
// ===== library types =====

TYPE "LHTTP_typeTLS"
   STRUCT
      validateServerIdentity : Bool;   // Validate the subjectAlternateName in the X.509-V3 certificate of the server to check the identity of the server
      serverCert : UDInt;   // ID of the X.509-V3 certificate (usually a CA certificate) that is used by the TLS client to validate the TLS server authentication. If this parameter is 0, the TLS client uses all (CA) certificates currently loaded in the client certificate store to validate the server authentication.
      clientCert : UDInt;   // ID of own X.509 V3 certificate
   END_STRUCT;
END_TYPE

// folder: GET

FUNCTION_BLOCK "LHTTP_Get"   // FB5, SCL
{ S7_Optimized_Access := 'TRUE' }
AUTHOR : AV
FAMILY : NET
VERSION : 0.1
   VAR_INPUT
      execute : Bool;   // Send HTTP request
      hwID : HW_ANY := 64;   // Hardware ID of Ethernet interface
      connID : CONN_OUC := 1;   // Unique connection ID
      url : String;   // URL, i.e. "http://www.siemens.com/simatic"
      data : String;   // Optional query parameters that are appended to URL, i.e. "lang=en&q=simatic"
      tls : "LHTTP_typeTLS";   // TLS certificates for secure connections (HTTPS), leave open for non-secure connections (HTTP)
   END_VAR
   VAR_OUTPUT
      done : Bool;   // HTTP request finished
      busy : Bool;   // Function is busy
      error : Bool;   // An error occured
      statusID : USInt;   // Specifies the source of the error
      status : Word;   // Specifies the error
      responseCode : UInt;   // HTTP response code
      length : UDInt;   // Length of received data
   END_VAR
   VAR_IN_OUT
      responseData : Array[*] of Char;   // Data received from HTTP server
   END_VAR
   VAR
      instTSend : TSEND_C;   // Instance of TSEND_C
      instTRcv : TRCV;   // Instance of TRCV
      instTimeout : TON_TIME;   // Time-out
      statDone : Bool;   // Static value for output 'done'
      statBusy : Bool;   // Static value for output 'busy'
      statError : Bool;   // Static value for output 'error'
      statStatusID : USInt;   // Static value for output 'statusID'
      statStatus : Word := 16#7000;   // Static value for output 'status'
      statFBState : USInt := 0;   // Current state in state machine
      statResponseCode : UInt;   // Static value for output 'responseCode'
      statEncoding : String;   // Transfer encoding of response from HTTP server
      statContentLength : UInt;   // Content length as specified in header of response
      statChunkLen : UInt;   // Remaining length of current chunk
      statRcvdLen : UDInt;   // Sum length of received data
      statLength : UDInt;   // Static value for output 'length'
      statParam : Struct   // Connection parameters
         isQDN : Bool;
         paramQDN : TCON_QDN_SEC;   // Connection parameters in form of QDN
         paramIP : TCON_IP_V4_SEC;   // Connection parameters in form of IP address
      END_STRUCT;
      statSend : Struct   // Parameters for instruction TSend_C
         connect : Bool;   // Establish and keep connection
         req : Bool;   // Send data
      END_STRUCT;
      statRequest : Struct   // GET request
         chars : Array[0..601] of Char;   // GET request (max. length: url (254) + data (254) + header (94)
         length : UInt;   // Length of GET request
      END_STRUCT;
      statTimeoutIn : Bool;   // Timeout
      statRcvBuffer : Array[0..1459] of Char;   // Temporary receive buffer; maximum segment size for TCP/IP is 1460
      statSizeRcvArray : UDInt;   // Size of receive buffer at parameter "responseData"
      statExecuteOld : Bool;   // Last cycle's value of input "execute"
   END_VAR
   VAR_TEMP
      tempLowerBound : DInt;   // Lower bound of receive buffer
      tempUrl : String;   // Copy of URL
      tempHost : String;   // Host part of URL
      tempPath : String;   // Path part of URL
      tempQuery : String;   // Query part of URL
      tempIndex : Int;   // Index for for loops
      tempPos : Int;   // General tag for positions
      tempLen : UInt;   // General tag for lengths
      tempRet : Word;   // General tag for return values
      tempString : String;   // General tag for strings
      tempExitLoop : Bool;   // Condition to exit REPEAT loop around state machine
      tempChunk : Struct   // Temporary tags for chunked encoding
         posData : UInt;   // Start position of data in current packet
         lenData : UInt;   // Length of data in current packet
         exitLoop : Bool;   // Condition to exit loop
      END_STRUCT;
   END_VAR
   VAR CONSTANT
      STATUS_DONE : Word := 16#0000;   // Job finished without errors
      STATUS_IDLE : Word := 16#7000;   // No job
      STATUS_FIRST_CALL : Word := 16#7001;   // First call after incoming new job (rising edge 'execute')
      STATUS_BUSY : Word := 16#7002;   // Intermediate call after job was started
      STATUS_BOUND_NOT_ZERO : Word := 16#8101;   // Lower bound of receive buffer is not 0
      STATUS_BUFFER_SIZE : Word := 16#8102;   // Receive buffer at parameter "responseData" too small
      STATUS_INVALID_URL : Word := 16#8103;   // Invalid URL
      STATUS_INVALID_HEADER : Word := 16#8104;   // Header of response is invalid
      STATUS_ENCODING_UNKNOWN : Word := 16#8105;   // Transfer encoding of response could not be detected or is unsupported
      STATUS_LENGTH_UNKNOWN : Word := 16#8106;   // Content length of response could not be detected
      STATUS_DECODING_FAILED : Word := 16#8107;   // Chunk encoded response could not be decoded
      STATUS_FORWARDING : Word := 16#8300;   // Server responded with forwarding message. Forwarding is not supported
      STATUS_TIMEOUT : Word := 16#8408;   // Time-out occurred
      STATUS_UNDEFINED_STATE : Word := 16#8600;   // Error due to an undefined state in state machine
      STATUS_ID_TSENDC : USInt := 1;   // Source of error is TSEND_C
      STATUS_ID_TRCV : USInt := 2;   // Source of error is TRCV
      STATUS_ID_MOVE_IDENTITY : USInt := 3;   // Source of error is MOVE_BLK_VARIANT for transfer encoding 'identity'
      STATUS_ID_MOVE_CHUNKED : USInt := 4;   // Source of error is MOVE_BLK_VARIANT for transfer encoding 'chunked'
      STATUS_ID_HTTP : USInt := 5;   // HTTP server signals error
      STATE_IDLE : USInt := 0;   // State no job
      STATE_INIT : USInt := 1;   // State initialization
      STATE_SEND : USInt := 2;   // State send request
      STATE_RCV : USInt := 3;   // State receive data
      TIMEOUT : Time := t#10s;   // Time to wait for response from server
      CRLF : String := '$R$L';   // ASCII characters for CRLF (carriage return & line feed)
      HEADER_END : String := '$R$L$R$L';   // End of HTTP header (double CRLF)
      LEN_CRLF : UInt := 2;   // Length of CRLF
   END_VAR
   // statParam.paramQDN.ConnPara.ActiveEstablished := true;
   // statParam.paramIP.ConnPara.ActiveEstablished := true;
BEGIN
   //=============================================================================
   // SIEMENS AG
   // (c)Copyright 2019
   //-----------------------------------------------------------------------------
   // Library:       LHTTP
   // Tested with:   CPU 1516-3 PN/DP V2.6
   // Engineering:   TIA Portal V15.1
   // Restrictions:  --
   // Requirements:  --
   // Functionality: Implements the HTTP GET method
   //-----------------------------------------------------------------------------
   // Change log table:
   // Version    Date         Expert in charge         Changes applied
   // 01.00.00   01.04.2019   Siemens Online Support   First released version
   //=============================================================================

   REGION INSTRUCTIONS
     IF (#statStatus <> #STATUS_IDLE) THEN // Only execute when FB is triggered to reduce system load
       // Connect and send
       IF #statParam.isQDN THEN // Call if host is a domain name
         #instTSend(REQ := #statSend.req,
                    CONT := #statSend.connect,
                    LEN := #statRequest.length,
                    CONNECT := #statParam.paramQDN,
                    DATA := #statRequest.chars);
       ELSE // Call if host is an IP address
         #instTSend(REQ := #statSend.req,
                    CONT := #statSend.connect,
                    LEN := #statRequest.length,
                    CONNECT := #statParam.paramIP,
                    DATA := #statRequest.chars);
       END_IF;

       // Receive
       #instTRcv(ID := #statParam.paramQDN.ConnPara.ID,
                 EN_R := #statFBState = #STATE_RCV,
                 LEN := 0,
                 ADHOC := true,
                 DATA := #statRcvBuffer);

       // Monitor time out
       #instTimeout(IN := #statTimeoutIn,
                    PT := #TIMEOUT);

       IF #instTimeout.Q THEN
         #statStatus := #STATUS_TIMEOUT;
       END_IF;
     END_IF;
   END_REGION

   REGION TRIGGERING
     IF (#execute = true) AND (#statExecuteOld = false) // Check if FB is triggered
       AND (#statStatus = #STATUS_IDLE)
     THEN // First call; initialize FB
       #statBusy := true;
       #statStatus := #STATUS_FIRST_CALL;
       #statFBState := #STATE_INIT;
     ELSIF (#statStatus = #STATUS_FIRST_CALL) THEN
       #statStatus := #STATUS_BUSY;
     END_IF;

     // Edge detection 'execute' input
     #statExecuteOld := #execute;
   END_REGION TRIGGERING

   IF (#statStatus = #STATUS_IDLE) THEN // Nothing to do -> End here to reduce "system load"
     RETURN;
   END_IF;

   REGION STATE_MACHINE
     // State machine is wrapped in REPEAT loop to make it possible to quickly exit state machine
     // in case of an error or to go through CASE multiple times within one cycle
     REPEAT
       #tempExitLoop := true; // Condition to exit loop is set per default

       CASE #statFBState OF // State machine of FB
         #STATE_IDLE: // No processing active (Note: this state must always be present and left empty)
           ;

         #STATE_INIT:
           REGION INIT
             // Get size of receive buffer
             #tempLowerBound := LOWER_BOUND(ARR := #responseData, DIM := 1);
             IF #tempLowerBound <> 0 THEN
               #statStatus := #STATUS_BOUND_NOT_ZERO;
               EXIT; // Exit loop immediately and output error
             ELSE
               #statSizeRcvArray := DINT_TO_UDINT(UPPER_BOUND(ARR := #responseData, DIM := 1)) + 1;
             END_IF;

             // Set connection parameters
             #statParam.paramQDN.ConnPara.InterfaceId := #hwID;
             #statParam.paramQDN.ConnPara.ID := #connID;
             #statParam.paramIP.ConnPara.InterfaceId := #hwID;
             #statParam.paramIP.ConnPara.ID := #connID;

             // Copy URL
             #tempUrl := #url;

             // Check if network protocol was specified to determine if connection should be secured
             IF #tempUrl[5] = 's' OR #tempUrl[5] = 'S' THEN // HTTPS
               #statParam.paramQDN.ActivateSecureConn := true;
               #statParam.paramQDN.ExtTLSCapabilities.%X0 := #tls.validateServerIdentity;
               #statParam.paramQDN.TLSServerCertRef := #tls.serverCert;
               #statParam.paramQDN.TLSClientCertRef := #tls.clientCert;
               #statParam.paramIP.ActivateSecureConn := true;
               #statParam.paramIP.ExtTLSCapabilities.%X0 := #tls.validateServerIdentity;
               #statParam.paramIP.TLSServerCertRef := #tls.serverCert;
               #statParam.paramIP.TLSClientCertRef := #tls.clientCert;
               // Delete network protocol from URL
               #tempUrl := DELETE(IN := #tempUrl, L := 8, P := 1);
             ELSE // HTTP
               #statParam.paramQDN.ActivateSecureConn := false;
               #statParam.paramIP.ActivateSecureConn := false;
               // Delete network protocol from URL if specified
               IF #tempUrl[5] = ':' THEN
                 #tempUrl := DELETE(IN := #tempUrl, L := 7, P := 1);
               END_IF;
             END_IF;

             // Determine if host is domain name or IP address
             #tempPos := CHAR_TO_INT(#tempUrl[1]);
             IF #tempPos >= CHAR_TO_INT('A') AND #tempPos <= CHAR_TO_INT('z') THEN // Host is a domain name
               #statParam.isQDN := true;
             ELSIF #tempPos >= CHAR_TO_INT('0') AND #tempPos <= CHAR_TO_INT('9') THEN // Host is an IP address
               #statParam.isQDN := false;
             ELSE // URL invalid
               #statStatus := #STATUS_INVALID_URL;
               EXIT; // Exit loop immediately
             END_IF;

             // Get host name and port
             #tempPos := FIND(IN1 := #tempUrl, IN2 := '/');
             IF #tempPos > 0 THEN // URL has a path after host name
               #tempHost := LEFT(IN := #tempUrl, L := #tempPos - 1);
               #tempPath := DELETE(IN := #tempUrl, L := #tempPos - 1, P := 1);
             ELSE
               #tempHost := #tempUrl;
               #tempPath := '/';
             END_IF;
             #tempPos := FIND(IN1 := #tempHost, IN2 := ':');
             IF #tempPos > 0 THEN // Port specified in URL
               #statParam.paramQDN.ConnPara.RemotePort := STRING_TO_UINT(DELETE(IN := #tempHost, L := #tempPos, P := 1));
               #statParam.paramIP.ConnPara.RemotePort := STRING_TO_UINT(DELETE(IN := #tempHost, L := #tempPos, P := 1));
               #tempHost := LEFT(IN := #tempHost, L := #tempPos - 1);
             ELSE // No port specified in URL, set default port
               IF #statParam.paramQDN.ActivateSecureConn OR #statParam.paramIP.ActivateSecureConn THEN
                 #statParam.paramQDN.ConnPara.RemotePort := 443;
                 #statParam.paramIP.ConnPara.RemotePort := 443;
               ELSE
                 #statParam.paramQDN.ConnPara.RemotePort := 80;
                 #statParam.paramIP.ConnPara.RemotePort := 80;
               END_IF;
             END_IF;

             IF #statParam.isQDN THEN // Host is a domain name
               #statParam.paramQDN.ConnPara.RemoteQDN := CONCAT(IN1 := #tempHost, IN2 := '.');
             ELSE // Host is an IP address
               #tempString := #tempHost;
               FOR #tempIndex := 1 TO 3 DO
                 #tempPos := FIND(IN1 := #tempString, IN2 := '.');
                 #statParam.paramIP.ConnPara.RemoteAddress.ADDR[#tempIndex] := UINT_TO_BYTE(STRING_TO_UINT(LEFT(IN := #tempString, L := #tempPos - 1)));
                 #tempString := DELETE(IN := #tempString, L := #tempPos, P := 1);
               END_FOR;
               #statParam.paramIP.ConnPara.RemoteAddress.ADDR[4] := UINT_TO_BYTE(STRING_TO_UINT(#tempString));
             END_IF;

             // Prepare query part of URL
             IF #data <> '' THEN // Parameter data is in use
               IF #data[1] = '?' OR #data[1] = '&' THEN
                 #tempQuery := DELETE(IN := #data, P := 1, L := 1);
               ELSE
                 #tempQuery := #data;
               END_IF;
               #tempPos := FIND(IN1 := #tempPath, IN2 := '?'); // Check if URL already contains query parameters
               IF #tempPos <> 0 THEN // URL already contains query parameters
                 #tempQuery := CONCAT(IN1 := '&', IN2 := #tempQuery); // Append query parameters with &
               ELSE // URL does not contain query parameters
                 #tempQuery := CONCAT(IN1 := '?', IN2 := #tempQuery); // Append query parameters with ?
               END_IF;
             END_IF;

             // Put together GET request
             // Strg_TO_Chars conversion is done several times to utilize maximum length of parameters url and data
             Strg_TO_Chars(Strg := CONCAT(IN1 := 'GET ', IN2 := #tempPath), // Path cannot be longer than 249 characters --> save to use CONCAT
                           pChars := 0,
                           Cnt => #tempLen,
                           Chars := #statRequest.chars);
             #tempPos := UINT_TO_INT(#tempLen);

             Strg_TO_Chars(Strg := #tempQuery,
                           pChars := #tempPos,
                           Cnt => #tempLen,
                           Chars := #statRequest.chars);
             #tempPos += UINT_TO_INT(#tempLen);

             Strg_TO_Chars(Strg := CONCAT(IN1 := ' HTTP/1.1$R$LHost: ', IN2 := #tempHost), // Host will not use all 254 characters --> save to use CONCAT
                           pChars := #tempPos,
                           Cnt => #tempLen,
                           Chars := #statRequest.chars);
             #tempPos += UINT_TO_INT(#tempLen);

             Strg_TO_Chars(Strg := '$R$LUser-Agent: SIMATIC S7-1500 (LHTTP)$R$LAccept: text/html$R$LAccept-Encoding: identity$R$LAccept-Charset: utf-8$R$L$R$L',
                           pChars := #tempPos,
                           Cnt => #tempLen,
                           Chars := #statRequest.chars);
             #statRequest.length := INT_TO_UINT(#tempPos) + #tempLen;

             #statSend.connect := true; // Connect
             #statSend.req := true; // Send request
             #statTimeoutIn := true; // Start timer
             #statFBState := #STATE_SEND;
           END_REGION

         #STATE_SEND: // Send data
           REGION SEND
             IF #instTSend.DONE THEN
               #statFBState := #STATE_RCV;
               // Stay in REPEAT loop to go directly to receive state
               // without waiting for next cycle so that no responses can be missed
               #tempExitLoop := false;
             ELSIF #instTSend.ERROR THEN
               #statStatusID := #STATUS_ID_TSENDC;
               #statStatus := #instTSend.STATUS;
             END_IF;
           END_REGION

         #STATE_RCV: // Wait for new data
           REGION RCV
             IF #instTRcv.NDR THEN

               REGION HEADER_EVAL
                 // Evaluate header if received packet is first packet
                 IF #statRcvdLen = 0 THEN
                   // Get response code
                   Chars_TO_Strg(Chars := #statRcvBuffer,
                                 pChars := 9,
                                 Cnt := 3,
                                 Strg => #tempString);
                   #statResponseCode := STRING_TO_UINT(#tempString);

                   // Exit loop immediately and output errror if response code shows errors or forwarding
                   IF #statResponseCode >= 400 THEN
                     #statStatusID := #STATUS_ID_HTTP;
                     #tempRet := ATH(IN := #tempString, N := 3, OUT => #statStatus); // Interpret response code as hexadecimal to integrate in status output
                     #statStatus := SHR(IN := #statStatus, N := 4);
                     #statStatus := 16#9000 OR #statStatus;
                     EXIT;
                   ELSIF #statResponseCode >= 300 THEN
                     #statStatus := #STATUS_FORWARDING;
                     EXIT;
                   END_IF;

                   // Get length of HTTP header
                   #tempLen := DINT_TO_UINT("LHTTP_FindStringInArray"(searchFor := #HEADER_END, searchIn := #statRcvBuffer) + LEN(#HEADER_END));

                   // Exit loop immediately and output errror if header end cannot be found
                   IF #tempLen = 0 THEN
                     #statStatus := #STATUS_INVALID_HEADER;
                     EXIT;
                   END_IF;

                   // Search header for content length
                   #tempRet := "LHTTP_ExtractStringFromArray"(textBefore := 'Content-Length: ',
                                                              textAfter := #CRLF,
                                                              extractedString => #tempString,
                                                              searchIn := #statRcvBuffer);

                   IF #tempRet = 0 THEN // Content length found
                     #statContentLength := STRING_TO_UINT(#tempString);
                     #statEncoding := 'identity';
                   ELSE // Can't detect content length, check if transfer encoding is 'chunked'
                     #tempPos := DINT_TO_INT("LHTTP_FindStringInArray"(searchFor := 'chunked', searchIn := #statRcvBuffer));

                     IF #tempPos >= 0 THEN
                       #statEncoding := 'chunked';
                     ELSE // Exit loop immediately and output error if content length nor transfer encoding can be detected
                       #statStatus := #STATUS_ENCODING_UNKNOWN;
                       EXIT;
                     END_IF;
                   END_IF;
                 END_IF;
               END_REGION

               REGION TE_IDENTITY
                 IF #statEncoding = 'identity' THEN // Transfer encoding is 'identity'
                   // Move data from buffer to output; tempLen contains header length during first packet, otherwise 0
                   #tempRet := INT_TO_WORD(MOVE_BLK_VARIANT(SRC := #statRcvBuffer,
                                                                                    COUNT := MIN(IN1 := #instTRcv.RCVD_LEN - #tempLen, IN2 := #statSizeRcvArray - #statRcvdLen), // Move as much as possible to output
                                                                                    SRC_INDEX := #tempLen,
                                                                                    DEST_INDEX := UDINT_TO_DINT(#statRcvdLen),
                                                                                    DEST => #responseData));

                   // Exit loop immediately and output error if data could not be moved
                   IF #tempRet <> 0 THEN
                     #statStatusID := #STATUS_ID_MOVE_IDENTITY;
                     #statStatus := #tempRet;
                     EXIT;
                   END_IF;

                   // Add length of received packet to sum; tempLen contains header length during first packet, otherwise 0
                   #statRcvdLen += #instTRcv.RCVD_LEN - #tempLen;

                   IF #statRcvdLen > #statSizeRcvArray THEN // Receive buffer too small
                     #statStatus := #STATUS_BUFFER_SIZE;
                     #statLength := #statContentLength; // Output required size of buffer
                   ELSIF #statRcvdLen >= #statContentLength THEN // Everything was received
                     #statStatus := #STATUS_DONE;
                     #statLength := #statRcvdLen;
                   END_IF;
                 END_IF;
               END_REGION

               REGION TE_CHUNKED
                 IF #statEncoding = 'chunked' THEN // Transfer encoding is 'chunked'

                   // Set position of chunk data
                   #tempChunk.posData := #tempLen; // tempLen contains header length during first packet, otherwise 0

                   REPEAT
                     #tempChunk.exitLoop := true; // Condition to exit loop is set per default

                     // Read length of chunk if received packet is first packet or a previous chunk was received completely
                     IF #statChunkLen = 0 THEN
                       // Extract hexadecimal length of chunk
                       Chars_TO_Strg(Chars := #statRcvBuffer,
                                     pChars := #tempChunk.posData,
                                     Cnt := 0,
                                     Strg => #tempString);
                       #tempPos := FIND(IN1 := #tempString, IN2 := #CRLF);
                       #tempRet := ATH(IN := #tempString, N := #tempPos - 1, OUT => #statChunkLen);
                       // Shift bits to the right depending on length of chunk size, since ATH is left aligned
                       #statChunkLen := SHR(IN := #statChunkLen, N := 4 * INT_TO_UINT(4 - (#tempPos - 1)));

                       // Move start position of data behind length indicator of chunk
                       #tempChunk.posData += INT_TO_UINT(#tempPos) + 1;

                       // Exit loop immediately and output error if length of chunk cannot be detected
                       IF #tempRet <> 0 THEN
                         #statStatus := #STATUS_DECODING_FAILED;
                         EXIT;
                       END_IF;
                     END_IF;

                     IF #statChunkLen = 0 THEN // Length was evaluated, chunk contains no data --> final chunk received
                       #statStatus := #STATUS_DONE;
                       #statLength := #statRcvdLen;
                     ELSE // Chunk contains data
                       // Evaluate length of received packet and set length of data accordingly
                       IF #instTRcv.RCVD_LEN = #tempChunk.posData + #statChunkLen + #LEN_CRLF THEN // Chunk was received entirely
                         #tempChunk.lenData := #statChunkLen - #LEN_CRLF; // Subtract line break to indicate end of chunk
                       ELSIF #instTRcv.RCVD_LEN < #tempChunk.posData + #statChunkLen + #LEN_CRLF THEN // Only part of chunk was received
                         #tempChunk.lenData := UDINT_TO_UINT(#instTRcv.RCVD_LEN) - #tempChunk.posData; // Output entire chunk
                       ELSIF #instTRcv.RCVD_LEN > #tempChunk.posData + #statChunkLen + #LEN_CRLF THEN // Current packet contains more data than indicated in chunk size
                         #tempChunk.lenData := #statChunkLen; // Subtract header and chunk length indicator
                         #tempChunk.exitLoop := false; // Execute loop again since packet contains more data
                       ELSE // Can't decode message
                         #statStatus := #STATUS_DECODING_FAILED;
                         EXIT;
                       END_IF;

                       // Move received data to output
                       #tempRet := INT_TO_WORD(MOVE_BLK_VARIANT(SRC := #statRcvBuffer,
                                                                                        COUNT := MIN(IN1 := #tempChunk.lenData, IN2 := #statSizeRcvArray - #statRcvdLen), // Move as much as possible to output
                                                                                        SRC_INDEX := #tempChunk.posData,
                                                                                        DEST_INDEX := UDINT_TO_DINT(#statRcvdLen),
                                                                                        DEST => #responseData));

                       // Exit loop immediately and output error if data could not be moved
                       IF #tempRet <> 0 THEN
                         #statStatusID := #STATUS_ID_MOVE_CHUNKED;
                         #statStatus := #tempRet;
                         EXIT;
                       END_IF;

                       // Move start position of data behind data of current chunk in case packet contains more data; only relevant if REPEAT loop is executed again
                       #tempChunk.posData += #tempChunk.lenData;

                       // Subtract length of data in current packet from remaining length of chunk and add to sum of received data
                       #statChunkLen -= #tempChunk.lenData;
                       #statRcvdLen += #tempChunk.lenData;

                       IF #statRcvdLen > #statSizeRcvArray THEN // Receive buffer too small
                         #statStatus := #STATUS_BUFFER_SIZE;
                         #statLength := #statRcvdLen; // Output required size of buffer according to so far received chunked messages
                       END_IF;
                     END_IF;
                   UNTIL (#tempChunk.exitLoop = true) END_REPEAT;
                 END_IF;
               END_REGION

             ELSIF #instTRcv.ERROR THEN
               #statStatusID := #STATUS_ID_TRCV;
               #statStatus := #instTRcv.STATUS;
             END_IF;
           END_REGION

         ELSE // Undefined state in state machine reached
           #statStatus := #STATUS_UNDEFINED_STATE;
       END_CASE;

     UNTIL (#tempExitLoop = true) END_REPEAT;
   END_REGION

   REGION OUTPUTS
     // Write outputs
     IF (#statStatus = #STATUS_DONE) AND (#statDone = false) THEN // Execution finished without errors
       #statDone := true;
       #statBusy := false;
       #statError := false;
       #statSend.connect := false;
       #statSend.req := false;
       #statTimeoutIn := false;
       #statFBState := #STATE_IDLE; // Switch state machine to "no processing"

     ELSIF (#statStatus.%X15 = true) AND (#statError = false) THEN // Error occurred (#statStatus is 16#8000 to 16#FFFF)
       #statDone := false;
       #statBusy := false;
       #statError := true;
       #statSend.connect := false;
       #statSend.req := false;
       #statTimeoutIn := false;
       #statFBState := #STATE_IDLE; // Switch state machine to "no processing"

     ELSIF (#execute = false) AND ((#statDone = true) OR (#statError = true)) THEN // Reset outputs
       #statDone := false;
       #statBusy := false;
       #statError := false;
       #statStatusID := 0;
       #statStatus := #STATUS_IDLE;
       #statResponseCode := 0;
       #statLength := 0;
       #statContentLength := 0;
       #statChunkLen := 0;
       #statEncoding := '';
       #statRcvdLen := 0;
       #statTimeoutIn := false;
     END_IF;

     // Write static values to outputs
     #done := #statDone;
     #busy := #statBusy;
     #error := #statError;
     #statusID := #statStatusID;
     #status := #statStatus;
     #responseCode := #statResponseCode;
     #length := #statLength;
   END_REGION OUTPUTS
END_FUNCTION_BLOCK

// folder: POST

FUNCTION_BLOCK "LHTTP_Post"   // FB6, SCL
{ S7_Optimized_Access := 'TRUE' }
AUTHOR : AV
FAMILY : NET
VERSION : 0.1
   VAR_INPUT
      execute : Bool;   // Send HTTP request
      hwID : HW_ANY := 64;   // Hardware ID of Ethernet interface
      connID : CONN_OUC := 1;   // Unique connection ID
      url : String;   // URL without scheme, i.e. "www.siemens.com/simatic"
      data : String;   // Data to transmit with POST request
      tls : "LHTTP_typeTLS";   // TLS certificates for secure connections (HTTPS), leave open for non-secure connections (HTTP)
   END_VAR
   VAR_OUTPUT
      done : Bool;   // HTTP request finished
      busy : Bool;   // Function is busy
      error : Bool;   // An error occured
      statusID : USInt;   // Specifies the source of the error
      status : Word;   // Specifies the error
      responseCode : UInt;   // HTTP response code
      length : UDInt;   // Length of received data
   END_VAR
   VAR_IN_OUT
      responseData : Array[*] of Char;   // Data received from HTTP server
   END_VAR
   VAR
      instTSend : TSEND_C;   // Instance of TSEND_C
      instTRcv : TRCV;   // Instance of TRCV
      instTimeout : TON_TIME;   // Time-out
      statDone : Bool;   // Static value for output 'done'
      statBusy : Bool;   // Static value for output 'busy'
      statError : Bool;   // Static value for output 'error'
      statStatusID : USInt;   // Static value for output 'statusID'
      statStatus : Word := 16#7000;   // Static value for output 'status'
      statFBState : USInt := 0;   // Current state in state machine
      statResponseCode : UInt;   // Static value for output 'responseCode'
      statEncoding : String;   // Transfer encoding of response from HTTP server
      statContentLength : UInt;   // Content length as specified in header of response
      statChunkLen : UInt;   // Remaining length of current chunk
      statRcvdLen : UDInt;   // Sum length f received packet
      statLength : UDInt;   // Static value for output 'length'
      statParam : Struct   // Connection parameters
         isQDN : Bool;
         paramQDN : TCON_QDN_SEC;   // Connection parameters in form of QDN
         paramIP : TCON_IP_V4_SEC;   // Connection parameters in form of IP address
      END_STRUCT;
      statSend : Struct   // Parameters for instruction TSend_C
         connect : Bool;   // Establish and keep connection
         req : Bool;   // Send data
      END_STRUCT;
      statRequest : Struct   // POST request
         chars : Array[0..667] of Char;   // POST request (max. length: url (254) + data (254) + header (157) + content-length (3)
         length : UInt;   // Length of POST request
      END_STRUCT;
      statTimeoutIn : Bool;   // Start timer
      statRcvBuffer : Array[0..1459] of Char;   // Temporary receive buffer; maximum segment size for TCP/IP is 1460
      statSizeRcvArray : UDInt;   // Size of receive buffer at parameter "responseData"
      statExecuteOld : Bool;   // Last cycle's value of input "execute"
   END_VAR
   VAR_TEMP
      tempLowerBound : DInt;   // Lower bound of receive buffer
      tempUrl : String;   // Copy of URL
      tempHost : String;   // Host part of URL
      tempPath : String;   // Path part of URL
      tempIndex : Int;   // Index for for loops
      tempPos : Int;   // General tag for positions
      tempLen : UInt;   // General tag for lengths
      tempRet : Word;   // General tag for return values
      tempString : String;   // General tag for strings
      tempExitLoop : Bool;   // Condition to exit REPEAT loop around state machine
      tempChunk : Struct   // Temporary tags for chunked encoding
         posData : UInt;   // Start position of data in current packet
         lenData : UInt;   // Length of data in current packet
         exitLoop : Bool;   // Condition to exit loop
      END_STRUCT;
   END_VAR
   VAR CONSTANT
      STATUS_DONE : Word := 16#0000;   // Job finished without errors
      STATUS_IDLE : Word := 16#7000;   // No job
      STATUS_FIRST_CALL : Word := 16#7001;   // First call after incoming new job (rising edge 'execute')
      STATUS_BUSY : Word := 16#7002;   // Intermediate call after job was started
      STATUS_BOUND_NOT_ZERO : Word := 16#8101;   // Status: Lower bound of receive buffer is not 0
      STATUS_BUFFER_SIZE : Word := 16#8102;   // Status: Receive buffer at parameter "data" too small
      STATUS_INVALID_URL : Word := 16#8103;   // Status: Invalid URL
      STATUS_INVALID_HEADER : Word := 16#8104;   // Header of response is invalid
      STATUS_ENCODING_UNKNOWN : Word := 16#8105;   // Transfer encoding of response could not be detected or is unsupported
      STATUS_LENGTH_UNKNOWN : Word := 16#8106;   // Content length of response could not be detected
      STATUS_DECODING_FAILED : Word := 16#8107;   // Chunk encoded response could not be decoded
      STATUS_FORWARDING : Word := 16#8300;   // Server responded with forwarding message. Forwarding is not supported
      STATUS_TIMEOUT : Word := 16#8408;   // Status: Time-out occurred
      STATUS_UNDEFINED_STATE : Word := 16#8600;   // Status: Error due to an undefined state in state machine
      STATUS_ID_TSENDC : USInt := 1;   // Source of error is TSEND_C
      STATUS_ID_TRCV : USInt := 2;   // Source of error is TRCV
      STATUS_ID_MOVE_IDENTITY : USInt := 3;   // Source of error is MOVE_BLK_VARIANT for transfer encoding 'identity'
      STATUS_ID_MOVE_CHUNKED : USInt := 4;   // Source of error is MOVE_BLK_VARIANT for transfer encoding 'chunked'
      STATUS_ID_HTTP : USInt := 5;   // HTTP server signals error
      STATE_IDLE : USInt := 0;   // State no job
      STATE_INIT : USInt := 1;   // State initialization
      STATE_SEND : USInt := 2;   // State send request
      STATE_RCV : USInt := 3;   // State receive data
      TIMEOUT : Time := t#10s;   // Time to wait for response from server
      CRLF : String := '$R$L';   // CRLF
      HEADER_END : String := '$R$L$R$L';   // End of HTTP header (double CRLF)
      LEN_CRLF : UInt := 2;   // Length of CRLF
   END_VAR
   // statParam.paramIP.ConnPara.ActiveEstablished := true;
   // statParam.paramQDN.ConnPara.ActiveEstablished := true;
   // statRequest.chars[1] := 'P';
   // statRequest.chars[2] := 'O';
   // statRequest.chars[3] := 'S';
   // statRequest.chars[4] := 'T';
   // statRequest.chars[5] := ' ';
BEGIN
   //=============================================================================
   // SIEMENS AG
   // (c)Copyright 2019
   //-----------------------------------------------------------------------------
   // Library:       LHTTP
   // Tested with:   CPU 1516-3 PN/DP V2.6
   // Engineering:   TIA Portal V15.1
   // Restrictions:  --
   // Requirements:  --
   // Functionality: Implements the HTTP POST method
   //-----------------------------------------------------------------------------
   // Change log table:
   // Version    Date         Expert in charge         Changes applied
   // 01.00.00   01.04.2019   Siemens Online Support   First released version
   //=============================================================================

   REGION INSTRUCTIONS
     IF (#statStatus <> #STATUS_IDLE) THEN // Only execute when FB is triggered to reduce system load
       // Connect and send
       IF #statParam.isQDN THEN // Call if host is a domain name
         #instTSend(REQ := #statSend.req,
                    CONT := #statSend.connect,
                    LEN := #statRequest.length,
                    CONNECT := #statParam.paramQDN,
                    DATA := #statRequest.chars);
       ELSE // Call if host is an IP address
         #instTSend(REQ := #statSend.req,
                    CONT := #statSend.connect,
                    LEN := #statRequest.length,
                    CONNECT := #statParam.paramIP,
                    DATA := #statRequest.chars);
       END_IF;

       // Receive
       #instTRcv(ID := #statParam.paramQDN.ConnPara.ID,
                 EN_R := #statFBState = #STATE_RCV,
                 LEN := 0,
                 ADHOC := true,
                 DATA := #statRcvBuffer);

       // Monitor time out
       #instTimeout(IN := #statTimeoutIn,
                    PT := #TIMEOUT);

       IF #instTimeout.Q THEN
         #statStatus := #STATUS_TIMEOUT;
       END_IF;
     END_IF;
   END_REGION

   REGION TRIGGERING
     IF (#execute = true) AND (#statExecuteOld = false) // Check if FB is triggered
       AND (#statStatus = #STATUS_IDLE)
     THEN // First call; initialize FB
       #statBusy := true;
       #statStatus := #STATUS_FIRST_CALL;
       #statFBState := #STATE_INIT;
     ELSIF (#statStatus = #STATUS_FIRST_CALL) THEN
       #statStatus := #STATUS_BUSY;
     END_IF;

     // Edge detection 'execute' input
     #statExecuteOld := #execute;
   END_REGION TRIGGERING

   IF (#statStatus = #STATUS_IDLE) THEN // Nothing to do -> End here to reduce "system load"
     RETURN;
   END_IF;

   REGION STATE_MACHINE
     // State machine is wrapped in REPEAT loop to make it possible to quickly exit state machine
     // in case of an error or to go through CASE multiple times within one cycle
     REPEAT
       #tempExitLoop := true; // Condition to exit loop is set per default

       CASE #statFBState OF // State machine of FB
         #STATE_IDLE: // No processing active (Note: this state must always be present and left empty)
           ;

         #STATE_INIT:
           REGION INIT
             // Get size of receive buffer
             #tempLowerBound := LOWER_BOUND(ARR := #responseData, DIM := 1);
             IF #tempLowerBound <> 0 THEN
               #statStatus := #STATUS_BOUND_NOT_ZERO;
               EXIT; // Exit loop immediately
             ELSE
               #statSizeRcvArray := DINT_TO_UDINT(UPPER_BOUND(ARR := #responseData, DIM := 1)) + 1;
             END_IF;

             // Set connection parameters
             #statParam.paramQDN.ConnPara.InterfaceId := #hwID;
             #statParam.paramQDN.ConnPara.ID := #connID;
             #statParam.paramIP.ConnPara.InterfaceId := #hwID;
             #statParam.paramIP.ConnPara.ID := #connID;

             // Copy URL
             #tempUrl := #url;

             // Check if network protocol was specified to determine if connection should be secured
             IF #tempUrl[5] = 's' OR #tempUrl[5] = 'S' THEN // HTTPS
               #statParam.paramQDN.ActivateSecureConn := true;
               #statParam.paramQDN.ExtTLSCapabilities.%X0 := #tls.validateServerIdentity;
               #statParam.paramQDN.TLSServerCertRef := #tls.serverCert;
               #statParam.paramQDN.TLSClientCertRef := #tls.clientCert;
               #statParam.paramIP.ActivateSecureConn := true;
               #statParam.paramIP.ExtTLSCapabilities.%X0 := #tls.validateServerIdentity;
               #statParam.paramIP.TLSServerCertRef := #tls.serverCert;
               #statParam.paramIP.TLSClientCertRef := #tls.clientCert;
               // Delete network protocol from URL
               #tempUrl := DELETE(IN := #tempUrl, L := 8, P := 1);
             ELSE // HTTP
               #statParam.paramQDN.ActivateSecureConn := false;
               #statParam.paramIP.ActivateSecureConn := false;
               // Delete network protocol from URL if specified
               IF #tempUrl[5] = ':' THEN
                 #tempUrl := DELETE(IN := #tempUrl, L := 7, P := 1);
               END_IF;
             END_IF;

             // Determine if host is domain name or IP address
             #tempPos := CHAR_TO_INT(#tempUrl[1]);
             IF #tempPos >= CHAR_TO_INT('A') AND #tempPos <= CHAR_TO_INT('z') THEN // Host is a domain name
               #statParam.isQDN := true;
             ELSIF #tempPos >= CHAR_TO_INT('0') AND #tempPos <= CHAR_TO_INT('9') THEN // Host is an IP address
               #statParam.isQDN := false;
             ELSE // URL invalid
               #statStatus := #STATUS_INVALID_URL;
               EXIT; // Exit loop immediately
             END_IF;

             // Get host name and port
             #tempPos := FIND(IN1 := #tempUrl, IN2 := '/');
             IF #tempPos > 0 THEN // URL has a path after host name
               #tempHost := LEFT(IN := #tempUrl, L := #tempPos - 1);
               #tempPath := DELETE(IN := #tempUrl, L := #tempPos - 1, P := 1);
             ELSE
               #tempHost := #tempUrl;
               #tempPath := '/';
             END_IF;
             #tempPos := FIND(IN1 := #tempHost, IN2 := ':');
             IF #tempPos > 0 THEN // Port specified in URL
               #statParam.paramQDN.ConnPara.RemotePort := STRING_TO_UINT(DELETE(IN := #tempHost, L := #tempPos, P := 1));
               #statParam.paramIP.ConnPara.RemotePort := STRING_TO_UINT(DELETE(IN := #tempHost, L := #tempPos, P := 1));
               #tempHost := LEFT(IN := #tempHost, L := #tempPos - 1);
             ELSE // No port specified in URL, set default port
               IF #statParam.paramQDN.ActivateSecureConn OR #statParam.paramIP.ActivateSecureConn THEN
                 #statParam.paramQDN.ConnPara.RemotePort := 443;
                 #statParam.paramIP.ConnPara.RemotePort := 443;
               ELSE
                 #statParam.paramQDN.ConnPara.RemotePort := 80;
                 #statParam.paramIP.ConnPara.RemotePort := 80;
               END_IF;
             END_IF;

             IF #statParam.isQDN THEN // Host is a domain name
               #statParam.paramQDN.ConnPara.RemoteQDN := CONCAT(IN1 := #tempHost, IN2 := '.');
             ELSE // Host is an IP address
               #tempString := #tempHost;
               FOR #tempIndex := 1 TO 3 DO
                 #tempPos := FIND(IN1 := #tempString, IN2 := '.');
                 #statParam.paramIP.ConnPara.RemoteAddress.ADDR[#tempIndex] := UINT_TO_BYTE(STRING_TO_UINT(LEFT(IN := #tempString, L := #tempPos - 1)));
                 #tempString := DELETE(IN := #tempString, L := #tempPos, P := 1);
               END_FOR;
               #statParam.paramIP.ConnPara.RemoteAddress.ADDR[4] := UINT_TO_BYTE(STRING_TO_UINT(#tempString));
             END_IF;

             // Put together POST request
             // Strg_TO_Chars conversion is done several times to utilize maximum length of parameters url and data
             Strg_TO_Chars(Strg := CONCAT(IN1 := 'POST ', IN2 := #tempPath), // Path cannot be longer than 249 characters --> save to use CONCAT
                           pChars := 0,
                           Cnt => #tempLen,
                           Chars := #statRequest.chars);
             #tempPos := UINT_TO_INT(#tempLen);

             Strg_TO_Chars(Strg := CONCAT(IN1 := ' HTTP/1.1$R$LHost: ', IN2 := #tempHost), // Host will not use all 254 characters --> save to use CONCAT
                           pChars := #tempPos,
                           Cnt => #tempLen,
                           Chars := #statRequest.chars);
             #tempPos += UINT_TO_INT(#tempLen);

             Strg_TO_Chars(Strg := '$R$LUser-Agent: SIMATIC S7-1500 (LHTTP)$R$LConnection: keep-alive$R$LAccept-Charset: utf-8$R$LContent-Encoding: identity$R$LContent-Type: text/plain$R$LContent-Length: ',
                           pChars := #tempPos,
                           Cnt => #tempLen,
                           Chars := #statRequest.chars);
             #tempPos += UINT_TO_INT(#tempLen);

             Strg_TO_Chars(Strg := CONCAT(IN1 := DELETE(IN := INT_TO_STRING(LEN(#data)), L := 1, P := 1), IN2 := #HEADER_END), // Calculate length of data
                           pChars := #tempPos,
                           Cnt => #tempLen,
                           Chars := #statRequest.chars);
             #tempPos += UINT_TO_INT(#tempLen);

             Strg_TO_Chars(Strg := #data,
                           pChars := #tempPos,
                           Cnt => #tempLen,
                           Chars := #statRequest.chars);
             #statRequest.length := INT_TO_UINT(#tempPos) + #tempLen;

             #statSend.connect := true; // Connect
             #statSend.req := true; // Send request
             #statTimeoutIn := true; // Start timer
             #statFBState := #STATE_SEND;
           END_REGION

         #STATE_SEND: // Send data
           REGION SEND
             IF #instTSend.DONE THEN
               #statFBState := #STATE_RCV;
               // Stay in REPEAT loop to go directly to receive state
               // without waiting for next cycle so that no responses can be missed
               #tempExitLoop := false;
             ELSIF #instTSend.ERROR THEN
               #statStatusID := #STATUS_ID_TSENDC;
               #statStatus := #instTSend.STATUS;
             END_IF;
           END_REGION

         #STATE_RCV: // Wait for new data
           REGION RCV
             IF #instTRcv.NDR THEN

               REGION HEADER_EVAL
                 // Evaluate header if received packet is first packet
                 IF #statRcvdLen = 0 THEN
                   // Get response code
                   Chars_TO_Strg(Chars := #statRcvBuffer,
                                 pChars := 9,
                                 Cnt := 3,
                                 Strg => #tempString);
                   #statResponseCode := STRING_TO_UINT(#tempString);

                   // Exit loop immediately and output errror if response code shows errors or forwarding
                   IF #statResponseCode >= 400 THEN
                     #statStatusID := #STATUS_ID_HTTP;
                     #tempRet := ATH(IN := #tempString, N := 3, OUT => #statStatus); // Interpret response code as hexadecimal to integrate in status output
                     #statStatus := SHR(IN := #statStatus, N := 4);
                     #statStatus := 16#9000 OR #statStatus;
                     EXIT;
                   ELSIF #statResponseCode >= 300 THEN
                     #statStatus := #STATUS_FORWARDING;
                     EXIT;
                   END_IF;

                   // Get length of HTTP header
                   #tempLen := DINT_TO_UINT("LHTTP_FindStringInArray"(searchFor := #HEADER_END, searchIn := #statRcvBuffer) + LEN(#HEADER_END));

                   // Exit loop immediately and output errror if header end cannot be found
                   IF #tempLen = 0 THEN
                     #statStatus := #STATUS_INVALID_HEADER;
                     EXIT;
                   END_IF;

                   // Search header for content length
                   #tempRet := "LHTTP_ExtractStringFromArray"(textBefore := 'Content-Length: ',
                                                              textAfter := #CRLF,
                                                              extractedString => #tempString,
                                                              searchIn := #statRcvBuffer);

                   IF #tempRet = 0 THEN // Content length found
                     #statContentLength := STRING_TO_UINT(#tempString);
                     #statEncoding := 'identity';
                   ELSE // Can't detect content length, check if transfer encoding is 'chunked'
                     #tempPos := DINT_TO_INT("LHTTP_FindStringInArray"(searchFor := 'chunked', searchIn := #statRcvBuffer));

                     IF #tempPos >= 0 THEN
                       #statEncoding := 'chunked';
                     ELSE // Exit loop immediately and output error if content length nor transfer encoding can be detected
                       #statStatus := #STATUS_ENCODING_UNKNOWN;
                       EXIT;
                     END_IF;
                   END_IF;
                 END_IF;
               END_REGION

               REGION TE_IDENTITY
                 IF #statEncoding = 'identity' THEN // Transfer encoding is 'identity'
                   // Move data from buffer to output; tempLen contains header length during first packet, otherwise 0
                   #tempRet := INT_TO_WORD(MOVE_BLK_VARIANT(SRC := #statRcvBuffer,
                                                                                    COUNT := MIN(IN1 := #instTRcv.RCVD_LEN - #tempLen, IN2 := #statSizeRcvArray - #statRcvdLen), // Move as much as possible to output
                                                                                    SRC_INDEX := #tempLen,
                                                                                    DEST_INDEX := UDINT_TO_DINT(#statRcvdLen),
                                                                                    DEST => #responseData));

                   // Exit loop immediately and output error if data could not be moved
                   IF #tempRet <> 0 THEN
                     #statStatusID := #STATUS_ID_MOVE_IDENTITY;
                     #statStatus := #tempRet;
                     EXIT;
                   END_IF;

                   // Add length of received packet to sum; tempLen contains header length during first packet, otherwise 0
                   #statRcvdLen += #instTRcv.RCVD_LEN - #tempLen;

                   IF #statRcvdLen > #statSizeRcvArray THEN // Receive buffer too small
                     #statStatus := #STATUS_BUFFER_SIZE;
                     #statLength := #statContentLength; // Output required size of buffer
                   ELSIF #statRcvdLen >= #statContentLength THEN // Everything was received
                     #statStatus := #STATUS_DONE;
                     #statLength := #statRcvdLen;
                   END_IF;
                 END_IF;
               END_REGION

               REGION TE_CHUNKED
                 IF #statEncoding = 'chunked' THEN // Transfer encoding is 'chunked'

                   // Set position of chunk data
                   #tempChunk.posData := #tempLen; // tempLen contains header length during first packet, otherwise 0

                   REPEAT
                     #tempChunk.exitLoop := true; // Condition to exit loop is set per default

                     // Read length of chunk if received packet is first packet or a previous chunk was received completely
                     IF #statChunkLen = 0 THEN
                       // Extract hexadecimal length of chunk
                       Chars_TO_Strg(Chars := #statRcvBuffer,
                                     pChars := #tempChunk.posData,
                                     Cnt := 0,
                                     Strg => #tempString);
                       #tempPos := FIND(IN1 := #tempString, IN2 := #CRLF);
                       #tempRet := ATH(IN := #tempString, N := #tempPos - 1, OUT => #statChunkLen);
                       // Shift bits to the right depending on length of chunk size, since ATH is left aligned
                       #statChunkLen := SHR(IN := #statChunkLen, N := 4 * INT_TO_UINT(4 - (#tempPos - 1)));

                       // Move start position of data behind length indicator of chunk
                       #tempChunk.posData += INT_TO_UINT(#tempPos) + 1;

                       // Exit loop immediately and output error if length of chunk cannot be detected
                       IF #tempRet <> 0 THEN
                         #statStatus := #STATUS_DECODING_FAILED;
                         EXIT;
                       END_IF;
                     END_IF;

                     IF #statChunkLen = 0 THEN // Length was evaluated, chunk contains no data --> final chunk received
                       #statStatus := #STATUS_DONE;
                       #statLength := #statRcvdLen;
                     ELSE // Chunk contains data
                       // Evaluate length of received packet and set length of data accordingly
                       IF #instTRcv.RCVD_LEN = #tempChunk.posData + #statChunkLen + #LEN_CRLF THEN // Chunk was received entirely
                         #tempChunk.lenData := #statChunkLen - #LEN_CRLF; // Subtract line break to indicate end of chunk
                       ELSIF #instTRcv.RCVD_LEN < #tempChunk.posData + #statChunkLen + #LEN_CRLF THEN // Only part of chunk was received
                         #tempChunk.lenData := UDINT_TO_UINT(#instTRcv.RCVD_LEN) - #tempChunk.posData; // Output entire chunk
                       ELSIF #instTRcv.RCVD_LEN > #tempChunk.posData + #statChunkLen + #LEN_CRLF THEN // Current packet contains more data than indicated in chunk size
                         #tempChunk.lenData := #statChunkLen; // Subtract header and chunk length indicator
                         #tempChunk.exitLoop := false; // Execute loop again since packet contains more data
                       ELSE // Can't decode message
                         #statStatus := #STATUS_DECODING_FAILED;
                         EXIT;
                       END_IF;

                       // Move received data to output
                       #tempRet := INT_TO_WORD(MOVE_BLK_VARIANT(SRC := #statRcvBuffer,
                                                                                        COUNT := MIN(IN1 := #tempChunk.lenData, IN2 := #statSizeRcvArray - #statRcvdLen), // Move as much as possible to output
                                                                                        SRC_INDEX := #tempChunk.posData,
                                                                                        DEST_INDEX := UDINT_TO_DINT(#statRcvdLen),
                                                                                        DEST => #responseData));

                       // Exit loop immediately and output error if data could not be moved
                       IF #tempRet <> 0 THEN
                         #statStatusID := #STATUS_ID_MOVE_CHUNKED;
                         #statStatus := #tempRet;
                         EXIT;
                       END_IF;

                       // Move start position of data behind data of current chunk in case packet contains more data; only relevant if REPEAT loop is executed again
                       #tempChunk.posData += #tempChunk.lenData;

                       // Subtract length of data in current packet from remaining length of chunk and add to sum of received data
                       #statChunkLen -= #tempChunk.lenData;
                       #statRcvdLen += #tempChunk.lenData;

                       IF #statRcvdLen > #statSizeRcvArray THEN // Receive buffer too small
                         #statStatus := #STATUS_BUFFER_SIZE;
                         #statLength := #statRcvdLen; // Output required size of buffer according to so far received chunked messages
                       END_IF;
                     END_IF;
                   UNTIL (#tempChunk.exitLoop = true) END_REPEAT;
                 END_IF;
               END_REGION

             ELSIF #instTRcv.ERROR THEN
               #statStatusID := #STATUS_ID_TRCV;
               #statStatus := #instTRcv.STATUS;
             END_IF;
           END_REGION

         ELSE // Undefined state in state machine reached
           #statStatus := #STATUS_UNDEFINED_STATE;
       END_CASE;

     UNTIL (#tempExitLoop = true) END_REPEAT;
   END_REGION

   REGION OUTPUTS
     // Write outputs
     IF (#statStatus = #STATUS_DONE) AND (#statDone = false) THEN // Execution finished without errors
       #statDone := true;
       #statBusy := false;
       #statError := false;
       #statSend.connect := false;
       #statSend.req := false;
       #statTimeoutIn := false;
       #statFBState := #STATE_IDLE; // Switch state machine to "no processing"

     ELSIF (#statStatus.%X15 = true) AND (#statError = false) THEN // Error occurred (#statStatus is 16#8000 to 16#FFFF)
       #statDone := false;
       #statBusy := false;
       #statError := true;
       #statSend.connect := false;
       #statSend.req := false;
       #statTimeoutIn := false;
       #statFBState := #STATE_IDLE; // Switch state machine to "no processing"

     ELSIF (#execute = false) AND ((#statDone = true) OR (#statError = true)) THEN // Reset outputs
       #statDone := false;
       #statBusy := false;
       #statError := false;
       #statStatusID := 0;
       #statStatus := #STATUS_IDLE;
       #statResponseCode := 0;
       #statLength := 0;
       #statContentLength := 0;
       #statChunkLen := 0;
       #statEncoding := '';
       #statRcvdLen := 0;
       #statTimeoutIn := false;
     END_IF;

     // Write static values to outputs
     #done := #statDone;
     #busy := #statBusy;
     #error := #statError;
     #statusID := #statStatusID;
     #status := #statStatus;
     #responseCode := #statResponseCode;
     #length := #statLength;
   END_REGION OUTPUTS
END_FUNCTION_BLOCK

// folder: Utilities

FUNCTION "LHTTP_ExtractStringFromArray" : Word   // FC2, SCL
{ S7_Optimized_Access := 'TRUE' }
VERSION : 0.1
   VAR_INPUT
      textBefore : String;   // Text before text that is extracted
      textAfter : String;   // Text after text that is extracted
   END_VAR
   VAR_OUTPUT
      extractedString : String;   // Extracted string
   END_VAR
   VAR_IN_OUT
      searchIn : Array[*] of Char;   // Array of Char to search in
   END_VAR
   VAR_TEMP
      tempLowerBound : DInt;   // Lower bound of given array
      tempNumElements : UDInt;   // Number of elements in given array
      tempPosInArray : DInt;   // Position in array during search
      tempLenTextBefore : Int;   // Length of text before
      tempPosTextBefore : DInt;   // Position of text before in array of Char
      tempLenTextAfter : Int;   // Length of text after
      tempPosTextAfter : Int;   // Position of text after in converted string
      tempString : String;   // Temporary string to work with
   END_VAR
   // Ret_Val : Return value; 16#0000: Successful, text was found, 16#9001: Unsuccessful, only start text was found, extracted String is filled with characters after start text, 16#9002: Unsuccessful, neither text was found
   VAR CONSTANT
      LEN_STRING : UInt := 254;   // Max. length of String
      STATUS_TEXT_FOUND : Word := 16#0000;   // Texts before and after were found
      STATUS_ONLY_START : Word := 16#9001;   // Only text before was found
      STATUS_NOTHING_FOUND : Word := 16#9002;   // Neither text was found
   END_VAR
BEGIN
   //=============================================================================
   // SIEMENS AG
   // (c)Copyright 2019
   //-----------------------------------------------------------------------------
   // Library:       LHTTP
   // Tested with:   CPU 1516-3 PN/DP V2.6
   // Engineering:   TIA Portal V15.1
   // Restrictions:  --
   // Requirements:  --
   // Functionality: Extracts a String specified by a text before and after
   //                from an array of Char
   //-----------------------------------------------------------------------------
   // Change log table:
   // Version    Date         Expert in charge         Changes applied
   // 01.00.00   01.04.2019   Siemens Online Support   First released version
   //=============================================================================

   // Initialization
   #tempPosTextBefore := 0;
   #tempPosTextAfter := 0;
   #tempLenTextBefore := LEN(#textBefore);
   #tempLenTextAfter := LEN(#textAfter);
   #extractedString := '';
   #LHTTP_ExtractStringFromArray := #STATUS_NOTHING_FOUND;

   // Get number of elements
   #tempPosInArray := #tempLowerBound := LOWER_BOUND(ARR := #searchIn, DIM := 1);
   #tempNumElements := DINT_TO_UDINT(UPPER_BOUND(ARR := #searchIn, DIM := 1) - #tempLowerBound + 1);


   // Search for text before until something was found
   REPEAT

     // Convert Chars to String
     Chars_TO_Strg(Chars  := #searchIn,
                   pChars := #tempPosInArray - #tempLowerBound, // Subtract offset since pChars is zero based
                   Cnt    := UDINT_TO_UINT(MIN(IN1 := #LEN_STRING, IN2 := #tempNumElements)),
                   Strg   => #tempString);

     // Search for text before
     #tempPosTextBefore := FIND(IN1 := #tempString, IN2 := #textBefore);

     // Text before was found
     IF #tempPosTextBefore > 0 THEN

       // Set position in array to end of text before
       #tempPosInArray += #tempPosTextBefore + #tempLenTextBefore - 1;

       // Create new string from end of text before
       Chars_TO_Strg(Chars  := #searchIn,
                     pChars := #tempPosInArray - #tempLowerBound, // Subtract offset since pChars is zero based
                     Cnt    := UDINT_TO_UINT(MIN(IN1 := #LEN_STRING, IN2 := #tempNumElements)),
                     Strg   => #tempString);

       // Find end of string to be extracted
       #tempPosTextAfter := FIND(IN1 := #tempString, IN2 := #textAfter);

       IF #tempPosTextAfter > 0 THEN // Shorten string if text after was found

         #extractedString := LEFT(IN := #tempString, L := #tempPosTextAfter - 1);
         #LHTTP_ExtractStringFromArray := #STATUS_TEXT_FOUND;
         EXIT;

       ELSE // Output whole string if text after was not found

         #extractedString := #tempString;
         #LHTTP_ExtractStringFromArray := #STATUS_ONLY_START;
         EXIT;

       END_IF;

     ELSE
       // Otherwise continue search in next string minus length of text before to ensure
       // keywords are not broken up at the end of a string and thus missed
       #tempPosInArray += UINT_TO_INT(#LEN_STRING) - #tempLenTextBefore;
     END_IF;

     // Repeat until end of array is reached
   UNTIL (#tempPosInArray > #tempNumElements) END_REPEAT;
END_FUNCTION

FUNCTION "LHTTP_ExtractStringFromArrayExt" : Word   // FC4, SCL
{ S7_Optimized_Access := 'TRUE' }
VERSION : 0.1
   VAR_INPUT
      textBefore : String;   // Text before text that is extracted
      textAfter : String;   // Text after text that is extracted
      includeBeforeAfter : Bool;   // If TRUE, texts before and after are included in the extracted string
      startPos : DInt;   // Position within array to start search from
   END_VAR
   VAR_OUTPUT
      extractedString : String;   // Extracted string
      position : DInt;   // Position (index) within the array where text begins
      length : Int;   // Length of text that was extracted
   END_VAR
   VAR_IN_OUT
      searchIn : Array[*] of Char;   // Array of Char to search in
   END_VAR
   VAR_TEMP
      tempLowerBound : DInt;   // Lower bound of given array
      tempNumElements : UDInt;   // Number of elements in given array
      tempPosInArray : DInt;   // Position in array during search
      tempLenTextBefore : Int;   // Length of text before
      tempPosTextBefore : DInt;   // Position of text before in array of Char
      tempLenTextAfter : Int;   // Length of text after
      tempPosTextAfter : Int;   // Position of text after in converted string
      tempString : String;   // Temporary string to work with
   END_VAR
   // Ret_Val : Return value; 16#0000: Successful, text was found, 16#9001: Unsuccessful, only start text was found, extracted String is filled with characters after start text, 16#9002: Unsuccessful, neither text was found
   VAR CONSTANT
      LEN_STRING : UInt := 254;   // Max. length of String
      STATUS_TEXT_FOUND : Word := 16#0000;   // Start text and end text were found
      STATUS_ONLY_START : Word := 16#9001;   // Only start text was found
      STATUS_NOTHING_FOUND : Word := 16#9002;   // Neither text was found
   END_VAR
BEGIN
   //=============================================================================
   // SIEMENS AG
   // (c)Copyright 2019
   //-----------------------------------------------------------------------------
   // Library:       LHTTP
   // Tested with:   CPU 1516-3 PN/DP V2.6
   // Engineering:   TIA Portal V15.1
   // Restrictions:  --
   // Requirements:  --
   // Functionality: Extracts a String specified by a text before and after
   //                from an array of Char with extended options
   //-----------------------------------------------------------------------------
   // Change log table:
   // Version    Date         Expert in charge         Changes applied
   // 01.00.00   01.04.2019   Siemens Online Support   First released version
   //=============================================================================

   // Initialization
   #tempPosInArray := #startPos;
   #tempPosTextBefore := 0;
   #tempPosTextAfter := 0;
   #tempLenTextBefore := LEN(#textBefore);
   #tempLenTextAfter := LEN(#textAfter);
   #position := -1;
   #length := 0;
   #extractedString := '';
   #LHTTP_ExtractStringFromArrayExt := #STATUS_NOTHING_FOUND;

   // Get number of elements
   #tempLowerBound := LOWER_BOUND(ARR := #searchIn, DIM := 1);
   #tempNumElements := DINT_TO_UDINT(UPPER_BOUND(ARR := #searchIn, DIM := 1) - #tempLowerBound + 1);

   // Search for text before until something was found
   REPEAT

     // Convert Chars to String
     Chars_TO_Strg(Chars := #searchIn,
                   pChars := #tempPosInArray - #tempLowerBound, // Subtract offset since pChars is zero based
                   Cnt := UDINT_TO_UINT(MIN(IN1 := #LEN_STRING, IN2 := #tempNumElements)),
                   Strg => #tempString);

     // Search for text before
     #tempPosTextBefore := FIND(IN1 := #tempString, IN2 := #textBefore);

     // Text before was found
     IF #tempPosTextBefore > 0 THEN

       // Set position in array to beginning or end of text before
       IF #includeBeforeAfter THEN
         #tempPosInArray += #tempPosTextBefore - 1;
       ELSE
         #tempPosInArray += #tempPosTextBefore + #tempLenTextBefore - 1;
       END_IF;

       // Create new string from beginning or end of text before
       Chars_TO_Strg(Chars := #searchIn,
                     pChars := #tempPosInArray - #tempLowerBound, // Subtract offset since pChars is zero based
                     Cnt := UDINT_TO_UINT(MIN(IN1 := #LEN_STRING, IN2 := #tempNumElements)),
                     Strg => #tempString);

       // Find end of string to be extracted
       #tempPosTextAfter := FIND(IN1 := #tempString, IN2 := #textAfter);

       IF #tempPosTextAfter > 0 THEN // Shorten string if text after was found

         IF #includeBeforeAfter THEN
           #length := #tempPosTextAfter + #tempLenTextAfter - 1;
         ELSE
           #length := #tempPosTextAfter - 1;
         END_IF;

         #position := #tempPosInArray;
         #extractedString := LEFT(IN := #tempString, L := #length);
         #LHTTP_ExtractStringFromArrayExt := #STATUS_TEXT_FOUND;
         EXIT;

       ELSE // Output whole string if text after was not found

         #extractedString := #tempString;
         #position := #tempPosInArray;
         #length := LEN(#tempString);
         #LHTTP_ExtractStringFromArrayExt := #STATUS_ONLY_START;
         EXIT;

       END_IF;

     ELSE
       // Otherwise continue search in next string minus length of text before to ensure
       // keywords are not broken up at the end of a string and thus missed
       #tempPosInArray += UINT_TO_INT(#LEN_STRING) - #tempLenTextBefore;
     END_IF;

     // Repeat until end of array is reached
   UNTIL (#tempPosInArray > #tempNumElements) END_REPEAT;
END_FUNCTION

FUNCTION "LHTTP_FindStringInArray" : DInt   // FC5, SCL
{ S7_Optimized_Access := 'TRUE' }
VERSION : 0.1
   VAR_INPUT
      searchFor : String;   // Text that is searched for
   END_VAR
   VAR_IN_OUT
      searchIn : Array[*] of Char;   // Array of Char to search in
   END_VAR
   VAR_TEMP
      tempLowerBound : DInt;   // Lower bound of given array
      tempNumElements : UDInt;   // Number of elements in given array
      tempLenSearchFor : Int;   // Length of text that is seached for
      tempPosInArray : DInt;   // Position in array during search (0-based)
      tempPosInString : Int;   // Position in working string during search
      tempString : String;   // Temporary string to work with
   END_VAR
   // Ret_Val : Position (index) of the first character of the text that is searched for within the array of Char
   VAR CONSTANT
      LEN_STRING : UInt := 254;   // Max. length of String
   END_VAR
BEGIN
   //=============================================================================
   // SIEMENS AG
   // (c)Copyright 2019
   //-----------------------------------------------------------------------------
   // Library:       LHTTP
   // Tested with:   CPU 1516-3 PN/DP V2.6
   // Engineering:   TIA Portal V15.1
   // Restrictions:  --
   // Requirements:  --
   // Functionality: Searches for a specified String within an array of Char
   //-----------------------------------------------------------------------------
   // Change log table:
   // Version    Date         Expert in charge         Changes applied
   // 01.00.00   01.01.2019   Siemens Online Support   First released version
   //=============================================================================

   // Initialization
   #tempPosInString := 0;
   #tempPosInArray := 0;
   #tempLenSearchFor := LEN(#searchFor);
   #LHTTP_FindStringInArray := -1;

   // Get number of elements
   #tempLowerBound := LOWER_BOUND(ARR := #searchIn, DIM := 1);
   #tempNumElements := DINT_TO_UDINT(UPPER_BOUND(ARR := #searchIn, DIM := 1) - #tempLowerBound + 1);

   // Search for beginning of text until something was found
   REPEAT

     // Convert Chars to String
     Chars_TO_Strg(Chars := #searchIn,
                   pChars := #tempPosInArray,
                   Cnt := UDINT_TO_UINT(MIN(IN1 := #LEN_STRING, IN2 := #tempNumElements)),
                   Strg => #tempString);

     // Search for text at beginning
     #tempPosInString := FIND(IN1 := #tempString, IN2 := #searchFor);

     // Keyword was found
     IF #tempPosInString > 0 THEN
       // Output position of string
       #LHTTP_FindStringInArray := #tempLowerBound + #tempPosInArray + #tempPosInString - 1;
       EXIT;
     ELSE
       // Otherwise continue search in next string minus length of text at beginning to ensure
       // keywords are not broken up at the end of a string and thus missed
       #tempPosInArray += UINT_TO_INT(#LEN_STRING) - #tempLenSearchFor;
     END_IF;

   UNTIL (#tempPosInString > 0) OR (#tempPosInArray > #tempNumElements) END_REPEAT;
END_FUNCTION

// ===== library: MasterCopy "LHTTP_Param" =====

DATA_BLOCK "LHTTP_Param"   // DB2
{ S7_Optimized_Access := 'TRUE' }
VERSION : 0.1
   VAR
      get : Struct
         execute : Bool;
         url : String;
         data : String;
         tls : "LHTTP_typeTLS";
         done : Bool;
         busy : Bool;
         error : Bool;
         statusID : USInt;
         status : Word;
         responseCode : UInt;
         length : UDInt;
      END_STRUCT;
      post : Struct
         execute : Bool;
         url : String;
         data : String;
         tls : "LHTTP_typeTLS";
      END_STRUCT;
   END_VAR
BEGIN
END_DATA_BLOCK